TYPE TcoInsightStatus_v_5_x_x : 
STRUCT
    ActionDescription : STRING(100);
    SignalStatus : TcoInsightSignalStates_v_5_x_x;
    CurrentJobName : STRING(100);
    CurrentJobNumber : INT := -1;
END_STRUCT
END_TYPE

(* stored: Version 1.1.0.1, ProductVersion 3.1.4024.11
   DUT TcoInsightStatus_v_5_x_x: Id {8761db8b-fe9a-0747-2397-36ef6a1e1714} *)
